FUNCTION_BLOCK FB_Tote_Subsystem EXTENDS FB_Generic
VAR_INPUT
	
END_VAR
VAR_OUTPUT
END_VAR
VAR
	tote_status_array 	AT%Q*	: ARRAY [0..99] OF ToteStatus;
	
	status					: MachineStatus := MachineStatus.STOPPED;	
	current_air_pressure	: REAL;	
	machine_control_cmd	 	: MachineControlCommand;
	
	cmd						: OrderToteCommand;
	
	ton1					: TON;

	ton_heart_beat			: TON;
	bReset_ads_heart_beat	: BOOL;
	bTest					: BOOL;
	
	machine_current_status	: E_PMLState;
	workflow1_status		: ToteSubsystemWorkflowStatus := ToteSubsystemWorkflowStatus.UNKNOWN;
	error1_status			: OrderToteErrorStatus := OrderToteErrorStatus.UNKNOWN;
	
	workflow2_status		: ToteSubsystemWorkflowStatus := ToteSubsystemWorkflowStatus.UNKNOWN;
	error2_status			: OrderToteErrorStatus := OrderToteErrorStatus.UNKNOWN;
	
	loading_tote			: ToteData;
	working1_tote			: ToteData;
	working2_tote			: ToteData;
	
	
	bInbound		: BOOL;
	bOutbound		: BOOL;
	bAbortInbound	: BOOL;
	bAbortOutbound	: BOOL;
	inboundToteParams_temp	: InboundToteParams;
	outboundToteParams_temp	: OutboundToteParams;
	abortToreParams_temp	: AbortToteRequestParams;

	A1	: INT;
	A2	: INT;
	iCase_abort	: INT;
END_VAR

SUPER^();
M_mapping();
IF sInstanceName='tote_1' THEN
	tote_status_array[0]	:= GVL.fb_loading.tote_status;
	tote_status_array[1]	:= GVL.fb_working1.tote_status;
	tote_status_array[2]	:= GVL.fb_working1.outboundTote_status;//outbound tote status form logtech
	machine_current_status	:= GVL.PackTags1.Status.StateCurrent;
END_IF
IF sInstanceName='tote_2' THEN
	tote_status_array[0]	:= GVL.fb_loading.tote_status;
	tote_status_array[1]	:= GVL.fb_working2.tote_status;
	tote_status_array[2]	:=  GVL.fb_working2.outboundTote_status;//outbound tote status form logtech
	machine_current_status	:= GVL.PackTags2.Status.StateCurrent;
END_IF

CASE machine_current_status OF
	ePMLState_Aborted,ePMLState_Aborting:
		status	:= MachineStatus.ERROR;
	ePMLState_Stopping:	
		status	:= MachineStatus.STOPPING;
	ePMLState_Stopped:
		status	:= MachineStatus.STOPPED;
	ePMLState_Resetting:	
		status	:= MachineStatus.RESETTING;
	ePMLState_Idle:	
		status	:= MachineStatus.READY;		
	ePMLState_Execute:	
		status	:= MachineStatus.RUNNING;			
END_CASE

IF bInbound THEN
	inboundToteParams_temp.source_id	:= ModelIdentifier.inbounding_position;
	inboundToteParams_temp.target_id	:= ModelIdentifier.working_position;
	inbound_tote_request(inbound_tote_params:=inboundToteParams_temp);
	bInbound	:= FALSE;
END_IF
IF bOutbound THEN
	outboundToteParams_temp.source_id	:= ModelIdentifier.working_position;
	outboundToteParams_temp.target_id	:= ModelIdentifier.outbound_position;	
	outbound_tote_request(outbound_tote_params:=outboundToteParams_temp);
	bOutbound	:= FALSE;
END_IF
IF bAbortInbound THEN
	abortToreParams_temp.source_id	:= ModelIdentifier.inbounding_position;
	abortToreParams_temp.target_id	:= ModelIdentifier.working_position;	
	abort_tote_request(abort_tote_request_params:=abortToreParams_temp);
	bAbortInbound	:= FALSE;
END_IF

IF bAbortOutbound THEN
	abortToreParams_temp.source_id	:= ModelIdentifier.working_position;
	abortToreParams_temp.target_id	:= ModelIdentifier.outbound_position;	
	abort_tote_request(abort_tote_request_params:=abortToreParams_temp);
	bAbortOutbound	:= FALSE;
END_IF

{attribute 'TcRpcEnable'}
METHOD abort_tote_request : UDINT//only response while awaiting
VAR_INPUT
	abort_tote_request_params : AbortToteRequestParams; // Struct containing data from the barcode scan	
END_VAR
abort_tote_request:=MethodCallReturnValue.DECLINED_BUSY;
IF sInstanceName='tote_1' THEN
	IF abort_tote_request_params.source_id=ModelIdentifier.inbounding_position AND abort_tote_request_params.target_id=ModelIdentifier.working_position THEN
		iCase_abort	:= 1;
	END_IF
	IF abort_tote_request_params.source_id=ModelIdentifier.working_position AND abort_tote_request_params.target_id=ModelIdentifier.outbound_position THEN
		iCase_abort	:= 2;
	END_IF		
	CASE iCase_abort OF
		1:
			IF GVL.fb_working1.tote_status=ToteStatus.AWAITING_INBOUND_AVAILABILITY THEN
				subData.Topic	:= E_Topics.WORKING1_ABORT_INBOUND;
				GVL.PubSubService.Publish(topic:=E_Topics.WORKING1_ABORT_INBOUND,data:= subData);
				abort_tote_request:= MethodCallReturnValue.ACCEPTED;
			ELSE
				abort_tote_request:= MethodCallReturnValue.DECLINED_ERROR;
			END_IF
		2:
			IF GVL.fb_working1.tote_status=ToteStatus.AWAITING_OUTBOUND_AVAILABILITY THEN
				subData.Topic	:= E_Topics.WORKING1_ABORT_OUTBOUND;
				GVL.PubSubService.Publish(topic:=E_Topics.WORKING1_ABORT_OUTBOUND,data:= subData);
				abort_tote_request:= MethodCallReturnValue.ACCEPTED;
			ELSE
				abort_tote_request:= MethodCallReturnValue.DECLINED_ERROR;
			END_IF	
		ELSE
			abort_tote_request:= MethodCallReturnValue.DECLINED_ERROR;
	END_CASE
END_IF

IF sInstanceName='tote_2' THEN
	IF abort_tote_request_params.source_id=ModelIdentifier.inbounding_position AND abort_tote_request_params.target_id=ModelIdentifier.working_position THEN
		iCase_abort	:= 1;
	END_IF
	IF abort_tote_request_params.source_id=ModelIdentifier.working_position AND abort_tote_request_params.target_id=ModelIdentifier.outbound_position THEN
		iCase_abort	:= 2;
	END_IF		
	CASE iCase_abort OF
		1:
			IF GVL.fb_working2.tote_status=ToteStatus.AWAITING_INBOUND_AVAILABILITY THEN
				subData.Topic	:= E_Topics.WORKING2_ABORT_INBOUND;
				GVL.PubSubService.Publish(topic:=E_Topics.WORKING2_ABORT_INBOUND,data:= subData);
				abort_tote_request:= MethodCallReturnValue.ACCEPTED;
			ELSE
				abort_tote_request:= MethodCallReturnValue.DECLINED_ERROR;
			END_IF
		2:
			IF GVL.fb_working2.tote_status=ToteStatus.AWAITING_INBOUND_AVAILABILITY THEN
				subData.Topic	:= E_Topics.WORKING2_ABORT_OUTBOUND;
				GVL.PubSubService.Publish(topic:=E_Topics.WORKING2_ABORT_OUTBOUND,data:= subData);
				abort_tote_request:= MethodCallReturnValue.ACCEPTED;
			ELSE
				abort_tote_request:= MethodCallReturnValue.DECLINED_ERROR;
			END_IF	
		ELSE
			abort_tote_request:= MethodCallReturnValue.DECLINED_ERROR;			
	END_CASE
END_IF
END_METHOD

{attribute 'TcRpcEnable'}
METHOD barcode_validation_request : UDINT
VAR_INPUT
	barcode_validation_request_params : BarcodeValidationRequestParams;
END_VAR
END_METHOD

{attribute 'TcRpcEnable'}
METHOD inbound_tote_request : UDINT
VAR_INPUT
	inbound_tote_params : InboundToteParams;
END_VAR
VAR	
	subData	: PubSubData;
END_VAR

IF sInstanceName='tote_1' THEN
//	IF NOT (((GVL.fb_working1.xLoading OR GVL.fb_working1.xInbound) AND GVL.fb_loading.xOutbound_woking1) OR 
//		GVL.fb_working1.tote_status=ToteStatus.LOADED OR GVL.fb_working1.xUnloading OR GVL.fb_working1.xOutbound) 
//	THEN//avoid cmd while inbounding or has tote
//		subData.Topic	:= E_Topics.WORKING1_INBOUND_TOTE;
//		GVL.PubSubService.Publish(topic:= E_Topics.WORKING1_INBOUND_TOTE,data:= subData);	
//	END_IF
	subData.Topic	:= E_Topics.WORKING1_INBOUND_TOTE;
	GVL.PubSubService.Publish(topic:= E_Topics.WORKING1_INBOUND_TOTE,data:= subData);
	A1	:= A1+1;	
END_IF
IF sInstanceName='tote_2' THEN
//	IF NOT (((GVL.fb_working2.xLoading OR GVL.fb_working2.xInbound) AND GVL.fb_loading.xOutbound_woking2) OR 
//		GVL.fb_working2.tote_status=ToteStatus.LOADED OR GVL.fb_working2.xUnloading OR GVL.fb_working2.xOutbound) 
//	THEN//avoid cmd while inbounding or has tote
//		subData.Topic	:= E_Topics.WORKING2_INBOUND_TOTE;
//		GVL.PubSubService.Publish(topic:= E_Topics.WORKING2_INBOUND_TOTE,data:= subData);
//	END_IF
	subData.Topic	:= E_Topics.WORKING2_INBOUND_TOTE;
	GVL.PubSubService.Publish(topic:= E_Topics.WORKING2_INBOUND_TOTE,data:= subData);
	A2	:= A2+1;
END_IF

//subData.Topic	:= E_Topics.RESET_WAITING_FOR_NEW_SPACE;
//GVL.PubSubService.Publish(topic:= E_Topics.RESET_WAITING_FOR_NEW_SPACE,data:= subData);
END_METHOD

{attribute 'TcRpcEnable'}
METHOD  init_tote_request : udint
VAR_INPUT
	init_tote_request_params : InitToteRequestParams;
END_VAR
init_tote_request:=1;
IF init_tote_request_params.source_id=ModelIdentifier.inbounding_position AND 
   init_tote_request_params.source_id=ModelIdentifier.working_position THEN 
  ;
     //MAIN.Machine.EM03.eState:=	E_WorkingStates.IDLE;				
//			MAIN.Machine.EM03.xLoading	:= FALSE;
//			MAIN.Machine.EM03.xUnloading	:= FALSE;
//			MAIN.Machine.EM03.xPerturbing := FALSE;
//			MAIN.Machine.EM03.xSwaping    := FALSE;
	 //MAIN.Machine.EM01.eState:=E_LoadingStates.IDLE;
END_IF  
IF init_tote_request_params.source_id=ModelIdentifier.working_position AND 
   init_tote_request_params.source_id=ModelIdentifier.outbound_position THEN 
;
    // MAIN.Machine.EM03.eState:=	E_WorkingStates.IDLE;				
//			MAIN.Machine.EM03.xLoading	:= FALSE;
//			MAIN.Machine.EM03.xUnloading	:= FALSE;
//			MAIN.Machine.EM03.xPerturbing := FALSE;
//			MAIN.Machine.EM03.xSwaping    := FALSE;
	// MAIN.Machine.EM04.eState:=E_UnloadingStates.IDLE;
END_IF  
init_tote_request:=0;
END_METHOD

METHOD M_mapping : BOOL
VAR_INPUT
END_VAR
END_METHOD

{attribute 'TcRpcEnable'}
METHOD outbound_tote_request : UDINT
VAR_INPUT
	outbound_tote_params : OutboundToteParams;	
END_VAR
VAR	
	subData	: PubSubData;
END_VAR
IF sInstanceName='tote_1' THEN
	IF NOT (GVL.fb_working1.xOutbound OR GVL.fb_working1.xInbound ) THEN//avoid cmd while outbounding
		subData.Topic	:= E_Topics.WORKING1_OUTBOUND_TOTE;
		GVL.PubSubService.Publish(topic:= E_Topics.WORKING1_OUTBOUND_TOTE,data:= subData);
	END_IF	
END_IF
IF sInstanceName='tote_2' THEN
	IF NOT (GVL.fb_working2.xOutbound OR GVL.fb_working2.xInbound ) THEN//avoid cmd while outbounding
		subData.Topic	:= E_Topics.WORKING2_OUTBOUND_TOTE;
		GVL.PubSubService.Publish(topic:= E_Topics.WORKING2_OUTBOUND_TOTE,data:= subData);
	END_IF
END_IF
END_METHOD

{attribute 'TcRpcEnable'}
METHOD perturb_tote_request : UDINT
VAR_INPUT
	perturb_tote_params : PerturbToteParams;	
END_VAR
IF //APP.Machine.CurrentStateEnum=E_PMLState.ePMLState_Execute 
//AND 
cmd=OrderToteCommand.DO_NOTHING
AND NOT MAIN.safety_1.bStop_button_unlock 
//AND NOT MAIN.safety_1.bBStop_button_unlock 
THEN
	cmd	:= OrderToteCommand.OPEN_BAG;
	perturb_tote_request:=0;
ELSE
	perturb_tote_request:=1;
END_IF
END_METHOD

{attribute 'TcRpcEnable'}
METHOD reset_tote_request : UDINT
VAR_INPUT
		
END_VAR
reset_tote_request	:= 1;

GVL.PackTags.Command.CntrlCmd:=1;

reset_tote_request	:= 0;
END_METHOD

{attribute 'TcRpcEnable'}
METHOD Setcmd : BOOL
VAR_INPUT
	orderToteCommand : OrderToteCommand;
END_VAR
cmd	:= orderToteCommand;
END_METHOD

{attribute 'TcRpcEnable'}
METHOD swap_tote_request : UDINT
VAR_INPUT
	swap_tote_params : SwapToteParams;	
END_VAR
IF //APP.Machine.CurrentStateEnum=E_PMLState.ePMLState_Execute 
//AND 
cmd=OrderToteCommand.DO_NOTHING
AND NOT MAIN.safety_1.bStop_button_unlock 
//AND NOT MAIN.safety_1.bBStop_button_unlock 
THEN
	cmd	:= OrderToteCommand.SWAP;
	swap_tote_request:=0;
ELSE
	swap_tote_request:=1;
END_IF
END_METHOD

END_FUNCTION_BLOCK

(* stored: Version 1.1.0.1, ProductVersion 3.1.4024.12
   POU FB_Tote_Subsystem: Id {18f3e813-8d9e-4f02-997f-31b8e26895c7}, SpecialFunc None
   Method abort_tote_request: Id {27f34e87-d12e-4bea-8d7e-cdf5426cb953}
   Method barcode_validation_request: Id {23a3884d-0782-4064-9104-e388dc1c5efc}
   Method inbound_tote_request: Id {62affe0d-84a6-41ac-aec8-cb5e0392a33c}
   Method init_tote_request: Id {a1f3fcdf-d013-416d-a1e1-2ac9181b9d6c}
   Method M_mapping: Id {541fb1a0-cd7a-4efb-8c21-3483a35c300d}
   Method outbound_tote_request: Id {60e6c187-39cd-4825-86c8-2f30debab9c2}
   Method perturb_tote_request: Id {a84801f4-88b7-49a6-af4b-2debbf0ff0a0}
   Method reset_tote_request: Id {77d9c51b-ed0b-4c37-8545-4a8fcb780fa9}
   Method Setcmd: Id {ba1f9cec-c3b0-46b8-a89b-cc046febc1a7}
   Method swap_tote_request: Id {f9f9c208-72c4-42e1-a02a-8ed4ea1b33b9} *)
